// TwinCAT 3 PLC project Timer_PLC
// ProgramVersion: 3.1.4020.10
// libraries:
//   Tc2_Standard, * (Beckhoff Automation GmbH)
//   Tc2_System, * (Beckhoff Automation GmbH)
//   Tc3_Interfaces, * (Beckhoff Automation GmbH)
//   Tc3_Module, * (Beckhoff Automation GmbH)
// project tree:
//   / PlcTask.TcTTO
//   POUs/ MAIN.TcPOU
// real-time tasks:
//   TASK PlcTask: cycle T#100us, priority 20, ADS port 350

CONFIGURATION Timer_PLC
    RESOURCE PLC ON TwinCAT3
        TASK PlcTask(INTERVAL := T#100us, PRIORITY := 20);
        PROGRAM MAIN WITH PlcTask : MAIN;
    END_RESOURCE
END_CONFIGURATION

// ---- POUs/MAIN.TcPOU
PROGRAM MAIN
VAR
	flag:		DWORD:=0;	//flag for noticing timer tick
	counter:	DWORD:=0;	//timer tick counter (1 = 100us = 0.1ms)
END_VAR

IF counter=9 THEN
	IF flag=0 THEN
		flag:=1;
	ELSE
		flag:=0;
	END_IF
	
	counter:=0;
ELSE
	counter:=counter+1;
END_IF

END_PROGRAM
